TYPE (* Primitive Type: String *)
  (* Version 1.0, 2023-02-23, Tim Hesse *)
  ROS2_std_msgs__String : STRUCT
    data : STRING;
  END_STRUCT;
END_TYPE
